//Tracking controller:
// Main handling of the control algorithm
// implements a state machine with states: init, idle, calcTrajectory, ready, driving
// links the different components of the control algorithm: control law, observer, trajectory, robot, camera... => Maybe more needed later e.g. filter 
// links to GW2 via the defined interface

PROGRAM TrackingController
VAR_INPUT
END_VAR
VAR_OUTPUT
END_VAR
VAR
	//declare objects
	observer 	: SimpleObserver;//Observer object
	controller	: SimpleStateFeedbackLaw;			//Control law object
	trajectory	: SimpleTrajectory;					//Trajectory Object
	robot		: Robot;							//link to physical I/O of roboter or simulation model of the roboter
	robotPoses 	AT%I*: ARRAY [1..8] OF RobotPose;	//input from camera
	
	state : ControllerState := ControllerState.init;//sets controller state
	
	CONTROL_ERROR_THRESH : LREAL := ;
	
	///////////////////////////////////////////////
	///////////// LINKS TO GW2  ///////////////////
	///////////////////////////////////////////////
	
	//inputs from GW2, uncomment and link when needed
	xBoEnable AT%I*: BOOL := FALSE;							// implemented, Freigabesignal für Fahrt, Roboter stoppt bei FALSE
	xIntMoveToEndPosition AT%I*: INT := 0;					// unused,		Anfahrt (in Sperrzone vor Tasche oder Ladestation) = 1, Fahrt = 0
	waypointList AT%I*: ARRAY[0..100] OF RobotPoseSimple;	// implemented, Wegpunktliste mit Roboter-Posen in globalen Koordinaten (x, y, theta)
	newWaypointListAvailable AT%I*: BOOL := FALSE;			// implemented, Status-Bit zur Signalisierung einer neuen WP-Liste
	
	//outputs to GW2, uncomment and link when needed
	yBoDriving AT%Q*: BOOL;									// implemented, TRUE, wenn Roboter fährt				
	yBoArrivedAtDestination AT%Q*:	BOOL := FALSE;			// implemented, TRUE, wenn Ziel erreicht, Ziel entspricht letzten gültigen WP
	yUintWaypointIndex AT%Q*: INT  := 0;						// implemented, COUNTER zur Anzeige, des Indexes des nächstes WP
	yRPposition AT%Q*: RobotPoseSimple;						// implemented, aktuelle Roboterposition, für Simulationszwecke
END_VAR

//robot disabled by default
robot.enable			:= FALSE;

//outputs to GW2
yBoDriving	 			:= robot.enable;
yRPposition 			:= observer.yObserverdPose;
yUintWaypointIndex 		:= trajectory.WPLidx;

//control algorithm state machine
CASE state OF
	ControllerState.init:
		//initilize objects and link them
		init();
		//go into idle
		state := ControllerState.idle;
	
	ControllerState.idle:
		//if new waypointlist go into trajectory calculation
		IF newWaypointListAvailable THEN
			state := ControllerState.calcTrajectory;
		END_IF
	
	ControllerState.calcTrajectory:
		//got new trajectory so not anymore at destination
		yBoArrivedAtDestination := FALSE;
		//calculate trajectory
		calculateTrajectory();
		//go into ready
		state := ControllerState.ready;
		
	
	ControllerState.ready:
		IF newWaypointListAvailable THEN
			//stop and calculate new trajectory
			state := ControllerState.calcTrajectory;
		ELSIF xBoEnable THEN
			state := ControllerState.driving;
		END_IF
	
	ControllerState.driving:
		IF newWaypointListAvailable THEN
			//stop and calculate new trajectory
			state := ControllerState.calcTrajectory;
		ELSIF trajectory.finished THEN
			//got back to idle and set arrived falg for GW2, method needed?
			yBoArrivedAtDestination := TRUE;
			state := ControllerState.idle;
		ELSIF xBoEnable THEN
			//do the driving
			drive();
		ELSE
			//if xBoEnable isn't set anymore go into ready and wait for it again
			state := ControllerState.ready;
		END_IF
END_CASE

//initilizing and linking of control algorithm individual components
//init observer
observer(xCameraPose := robotPoses[Var_HAWIno.Robot_Number],	//extraxt roboter coordinates based on roboter number
		 xVxRobot    := robot.vXfromRobot,						//link x-velocity with measured velocity
		 xVyRobot    := robot.vYfromRobot,						//link y-velocity with measured velocity
		 xOmegaRobot    := robot.vThetaFromRobot);				//link theta-velocity with measured velocity

//init controller and link to observer
controller(xRobotPose 		:= observer.yObserverdPose,			//pass controller the observerd roboter pose
		   xRobotPoseRef	:= trajectory.referencePose);		//pass controller the reference position for the next cycle comming from the trajectory

//transform control inputs into robot coordinates and pass them to the robot
//pass enable signal to robot
World2Robot(
			vx_world := controller.vXrobot,						//controller outputs vXref in world coordinates
			vy_world := controller.vYrobot,						//controller outputs vYref in world coordinates
			omega_world := controller.omegaRobot,				//controller outputs vThetaRef in world coordinates
			theta := observer.yObserverdPose.theta,				//observed theta for transoformation in robot coordinates
			vx_robot => robot.vXref,							//vXref in robot coordinates are passed to robot as control output
			vy_robot => robot.vYref,							//vYref in robot coordinates are passed to robot as control output
			omega_robot => robot.vThetaRef						//vThetaref in robot coordinates are passed to robot as control output
);

//trajectory object
trajectory(
	currentPose 	:= observer.yObserverdPose,					//Current implementation needs observed pose for distance calculation, TODO: check if needed for final implemenation
	referencePose 	=> controller.xRobotPoseRef					//outputs reference pose to controller
);


// to do:
IF trajectory.finished AND controller.reachedReference THEN
	yBoArrivedAtDestination := TRUE;
END_IF




//needs to be called so that the velocities will be written to motor drives
robot();

METHOD calculateTrajectory : BOOL
VAR_INPUT
END_VAR
trajectory.setWaypointList(waypointList);
END_METHOD

METHOD drive : BOOL
VAR_INPUT
END_VAR
robot.enable := TRUE;
END_METHOD

METHOD init : BOOL
VAR_INPUT
END_VAR
VAR
END_VAR
END_METHOD

END_PROGRAM

(* stored: Version 1.1.0.1, ProductVersion 3.1.4024.11
   POU TrackingController: Id {012ed989-ad00-4074-8a95-3f6b38ed2b93}, SpecialFunc None
   Method calculateTrajectory: Id {8f230d49-0c59-4087-8372-938452edcf61}
   Method drive: Id {d4cf0706-755e-4b45-b3e9-0b9f8575bd33}
   Method init: Id {0d1b690b-7302-4509-955c-4b8bf838eebc} *)
